// Acknowledgement-Examples.
// > One object per demonstrated 'AlarmMode'.
// > See "FB_BA_EC01" to view decleared event classes.
// [Hint]
// > All reference-variables are implemented to ease monitoring of relevant variables.
// > show the possibility to acknowledge BA objects assigned to a specific event class.
FUNCTION_BLOCK FB_Evt_Ack EXTENDS FB_BA_View
VAR               
	{region 'General'}
		bAlm_Test						: BOOL;																						// Trigger alarm for testing.
		bAlm_AckAll						: REFERENCE TO BOOL							REF= THIS^.bAcknowledgeRm;						// Acknowledge all test objects.
		bAlm_AckMode					: POINTER TO BOOL							:= ADR(XBA_Param.eEvtMgmt_AckMode);				// Used reset mode (See parameter description for more details)
	{endregion}
		 
	{region 'Simple'}
		// Intention:					Alarm that automatically disappears.
		// State on active alarm:		- "bEvent = TRUE'
		//								- "stAckedTransitions = [FALSE,true,true]'
		// State when disappeared:		- "bEvent = false'
		//								- "stAckedTransitions = [true,true,true]'
		AlmSimple_Ack					: REFERENCE TO BOOL							REF= AlmSimple.bAcknowledgeRm;
		AlmSimple_Indicated				: BOOL;
		AlmSimple_Event					: REFERENCE TO BOOL							REF= AlmSimple.bEvent;
		AlmSimple						: FB_BA_BI_Raw := (
											iParent									:= THIS^,
											sInactiveText							:= 'Normal',
											sActiveText								:= 'Alarm',
											nEventClassID							:= MyECIDs.AlmSmpl);
	{endregion}
	{region 'Standard'}
		// Intention:					Alarm that is just indicated (by acknowledge transition) when disappeared.
		// State on active alarm:		- "bEvent = TRUE'
		//								- "stAckedTransitions = [FALSE,true,true]'
		// State when disappeared:		- "bEvent = false'
		//								- "stAckedTransitions = [FALSE,true,true]'
		// State after acknowledgement:	- "bEvent = false'
		//								- "stAckedTransitions = [true,true,true]'
		AlmStandard_Ack					: REFERENCE TO BOOL							REF= AlmStandard.bAcknowledgeRm;
		AlmStandard_Indicated			: BOOL;
		AlmStandard_Event				: REFERENCE TO BOOL							REF= AlmStandard.bEvent;
		AlmStandard						: FB_BA_BI_Raw := (
											iParent									:= THIS^,
											sInactiveText							:= 'Normal',
											sActiveText								:= 'Alarm',
											nEventClassID							:= MyECIDs.AlmStd);	
	{endregion}
	{region 'Extended'}
		// Intention:					Alarm that is indicated (by acknowledge transition) and hold when disappeared.
		//								The 'bEvent' is released when an additional reset has been triggered.
		// State on active alarm:		- "bEvent = TRUE'
		//								- "stAckedTransitions = [FALSE,true,FALSE]'
		// State when disappeared:		- "bEvent = TRUE'
		//								- "stAckedTransitions = [FALSE,true,FALSE]'
		// State after acknowledgement:	- "bEvent = TRUE'
		//								- "stAckedTransitions = [true,true,FALSE]'
		// State after reset:			- "bEvent = false'
		//								- "stAckedTransitions = [true,true,true]'
		AlmExtended_Ack					: REFERENCE TO BOOL							REF= AlmExtended.bAcknowledgeRm;
		AlmExtended_Indicated			: BOOL;
		AlmExtended_Event				: REFERENCE TO BOOL							REF= AlmExtended.bEvent;
		AlmExtended						: FB_BA_BI_Raw := (
											iParent									:= THIS^,
											sInactiveText							:= 'Normal',
											sActiveText								:= 'Alarm',
											nEventClassID							:= MyECIDs.AlmExt);	
	{endregion}	
		 
	{region 'Acknowledge event class'}	
		// Intention:					Acknowledge all objects that reference a specific event class.
		nEventClassID					: UINT										:= 0;			// Enter ID of event class to acknowledge.
	{endregion}
		 
END_VAR

SUPER^();

AlmSimple(bRawVal:=bAlm_Test);
AlmSimple_Indicated := (NOT AlmSimple.stAckedTransitions.bToOffnormal);
AlmStandard(bRawVal:=bAlm_Test);
AlmStandard_Indicated := (NOT AlmStandard.stAckedTransitions.bToOffnormal);
AlmExtended(bRawVal:=bAlm_Test);
AlmExtended_Indicated := (NOT AlmExtended.stAckedTransitions.bToOffnormal);

IF (nEventClassID <> 0) THEN
	F_AcknowledgeEventClass(nEventClassID);
	nEventClassID := 0;
END_IF

// Intention:			Illustrate how to recognize changed events.
METHOD PROTECTED OnObjectEventChange
VAR_INPUT
	iObject				: I_BA_EventObject;
	bNotifyParents		: BOOL				:= TRUE;
END_VAR
SUPER^.OnObjectEventChange(iObject, bNotifyParents);

// Sample 1) Evaluate current event state:
CASE (iObject.EventIcon.eState) OF
	E_BA_EventIconState.eGoneAcked,
	E_BA_EventIconState.ePresentAcked:
		iObject.LogMsg.Show(ADSLOG_MSGTYPE_HINT, 'OOEC06', 'Object acknowledged.', TRUE);
END_CASE

// Sample 2) Compare actual event state to previous event state:
IF (iObject.LastEventIcon.eState < iObject.EventIcon.eState) THEN
	; // State intensed...
ELSE
	; // State softened...
END_IF
END_METHOD

END_FUNCTION_BLOCK

(* stored: Version 1.1.0.1, ProductVersion 3.1.4024.12
   POU FB_Evt_Ack: Id {fbc947ed-fc04-4bb0-b954-ae66748fd31d}, SpecialFunc None
   Folder [Protected] Events: Id {4aff504b-1474-44a7-b295-050cdde9c749}
   Method OnObjectEventChange: Id {20aa6ae7-33a9-417c-8eaa-995d30bdb29f} *)
